// TwinCAT 3 PLC project PRG_B_IO
// Title: B_IO
// Company: RafalOS
// Author: Rafał Osajda
// ProjectVersion: 0.0.0.5
// ProgramVersion: 3.1.4024.0
// libraries:
//   B_Base, * (RafalOS)
//   Tc2_Standard, * (Beckhoff Automation GmbH)
//   Tc2_System, * (Beckhoff Automation GmbH)
//   Tc3_Module, * (Beckhoff Automation GmbH)
// project tree:
//   / PlcTask.TcTTO
//   POUs Compilation/ PRG_Compilation.TcPOU
//   POUs/Electrovalve/ E_ElectrovalveAction.TcDUT, E_ElectrovalveType.TcDUT, FB_Electrovalve.TcPOU, FB_Electrovalve_3on2_NC.TcPOU, FB_Electrovalve_3on2_NO.TcPOU, FB_Electrovalve_5on2_1Coil.TcPOU, FB_Electrovalve_5on2_2Coil.TcPOU, FB_Electrovalve_5on3_2Coil_Vented.TcPOU, FB_Electrovalve_5on3_2Coil_Infected.TcPOU, ITF_Electrovalve.TcIO, ITF_Electrovalve_HMI_Init.TcIO, ITF_Electrovalve_HMI_Connector.TcIO
//   POUs/Sensor/ E_SensorType.TcDUT, FB_Sensor.TcPOU, FB_Sensor_NC.TcPOU, FB_Sensor_NO.TcPOU, FB_Sensor_NO_2InRow.TcPOU, ITF_Sensor.TcIO, ITF_Sensor_HMI_Init.TcIO, ITF_Sensor_HMI_Connector.TcIO
//   POUs/LampkaRozszerzona/ FB_LampBlinking.TcPOU, ITF_LampBlinking.TcIO
//   POUs/Lampka/ FB_Lamp.TcPOU, ITF_Lamp.TcIO
//   POUs/Przyciski/ FB_Button.TcPOU, FB_Button_NC.TcPOU, FB_Button_NO.TcPOU, ITF_Button.TcIO
// real-time tasks:
//   TASK PlcTask: cycle T#10ms, priority 20, ADS port 350

CONFIGURATION PRG_B_IO
    RESOURCE PLC ON TwinCAT3
        TASK PlcTask(INTERVAL := T#10ms, PRIORITY := 20);
        PROGRAM PRG_Compilation WITH PlcTask : PRG_Compilation;
    END_RESOURCE
END_CONFIGURATION

// ---- POUs/Electrovalve/E_ElectrovalveAction.TcDUT
{attribute 'qualified_only'}
{attribute 'strict'}
TYPE E_ElectrovalveAction :
(
	e_EV_Out4_Deactive 	:= 1,
	e_EV_OUT4_Active	:= 2,
	e_EV_Out2_Deactive 	:= 3,
	e_EV_Out2_Active	:= 4,
	e_EV_ToStart		:= 5,
	e_EV_ToEnd			:= 6,
	e_EV_Stop			:= 7,
	e_EV_Reset			:= 8,
	e_EV_Active			:= 9,
	e_EV_Deactive		:= 10
);
END_TYPE

// ---- POUs/Electrovalve/E_ElectrovalveType.TcDUT
{attribute 'qualified_only'}
{attribute 'strict'}
TYPE E_ElectrovalveType :
(
	NC_3na2 	:= 0,
	NO_3na2		:= 1,
	C1_5na2		:= 2,
	C2_5na2		:= 3,
	C2_5na3O	:= 4,	//odpowietrzony
	C2_5na3Z	:= 5	//Zapowietrzony
);
END_TYPE

// ---- POUs/Sensor/E_SensorType.TcDUT
{attribute 'qualified_only'}
{attribute 'strict'}
TYPE E_SensorType :
(
	NO 		:= 0,
	NC		:= 1,
	NOx2	:= 2
);
END_TYPE

// ---- POUs/Sensor/ITF_Sensor.TcIO
(*			
	EVERDE sp. z o.o.
	Rafał Osajda		22.01.2025		TC 4026.13		wer. 0.0.0.1
	B_Baza dla czujników binarnych 	
*)
INTERFACE ITF_Sensor EXTENDS ITF_BaseComponent

(*			
	EVERDE sp. z o.o.
	Rafał Osajda		05.02.2025		TC 4026.13		wer. 0.0.0.1
	Zwraca aktualny stan czujnika
*)
METHOD IsActive : BOOL
END_METHOD

END_INTERFACE

// ---- POUs/Sensor/ITF_Sensor_HMI_Init.TcIO
(*			
	EVERDE sp. z o.o.
	Rafał Osajda		21.08.2025		TC 4024.66
	Interfejs łaczący na potrzeby przekazania do elementu
*)
INTERFACE ITF_Sensor_HMI_Init EXTENDS ITF_BaseComponent, ITF_Sensor_HMI_Connector

END_INTERFACE

// ---- POUs/Sensor/ITF_Sensor_HMI_Connector.TcIO
INTERFACE ITF_Sensor_HMI_Connector EXTENDS ITF_BaseComponent_HMI_Connector

METHOD PUBLIC GetSensorType : E_SensorType
VAR_INPUT
END_VAR
END_METHOD

METHOD PUBLIC GetSensorTypeToString : STRING
END_METHOD

(*			
	EVERDE sp. z o.o.
	Rafał Osajda		05.02.2025		TC 4026.13		wer. 0.0.0.1
	Zwraca aktualny stan czujnika
*)
METHOD IsActive : BOOL
END_METHOD

END_INTERFACE

// ---- POUs/Electrovalve/ITF_Electrovalve.TcIO
(*
	RJM Maszyny sp. z o.o.
	autor 	: Rafał Osajda
	data	: 21.02.2024
	TC		: 3.1 4024.54
	wersja	: 0.0.1.0	: pełna obsługa

	Obsługa elektrozaworu do sterowania siłownikiem pneumatycznym
*)
INTERFACE ITF_Electrovalve EXTENDS ITF_BaseComponent

(*
	RJM Maszyny sp. z o.o.
	autor 	: Rafał Osajda
	data	: 21.02.2024
	TC		: 3.1 4024.54
	wersja	: 0.0.1.0	: pełna obsługa

	Ustawienie odpowiednich wyjść
*)
METHOD Contol : BOOL
VAR_INPUT
	eAction									: E_ElectrovalveAction;
END_VAR
END_METHOD

END_INTERFACE

// ---- POUs/Electrovalve/ITF_Electrovalve_HMI_Init.TcIO
(*			
	EVERDE sp. z o.o.
	Rafał Osajda		21.08.2025		TC 4024.66
	Interfejs łaczący na potrzeby przekazania do elementu
*)
INTERFACE ITF_Electrovalve_HMI_Init EXTENDS ITF_BaseComponent, ITF_Electrovalve_HMI_Connector

END_INTERFACE

// ---- POUs/Electrovalve/ITF_Electrovalve_HMI_Connector.TcIO
INTERFACE ITF_Electrovalve_HMI_Connector EXTENDS ITF_BaseComponent_HMI_Connector

METHOD PUBLIC GetElectrovalveType : E_ElectrovalveType
VAR_INPUT
END_VAR
END_METHOD

METHOD PUBLIC GetElectrovalveTypeToString : STRING
END_METHOD

METHOD IsActiveCoilA : BOOL
VAR_INPUT
END_VAR
END_METHOD

METHOD IsActiveCoilB : BOOL
VAR_INPUT
END_VAR
END_METHOD

END_INTERFACE

// ---- POUs/LampkaRozszerzona/ITF_LampBlinking.TcIO
INTERFACE ITF_LampBlinking EXTENDS ITF_Lamp

(*			
	EVERDE sp. z o.o.
	Rafał Osajda		31.01.2025		TC 4026.13		wer. 0.0.0.1
	Sterowanie działem ipulsatora 
*)
METHOD PUBLIC SetBlink
VAR_INPUT
	bIN				: bool;
END_VAR
END_METHOD

(*			
	EVERDE sp. z o.o.
	Rafał Osajda		31.01.2025		TC 4026.13		wer. 0.0.0.1
	Ustawia czas zgaszonej lampki
*)
METHOD PUBLIC SetTimeOff
VAR_INPUT
	rIN					: REAL;
END_VAR
END_METHOD

(*			
	EVERDE sp. z o.o.
	Rafał Osajda		31.01.2025		TC 4026.13		wer. 0.0.0.1
	
*)
METHOD PUBLIC SetTimeOn
VAR_INPUT
	rIN						: REAL;
END_VAR
END_METHOD

METHOD PUBLIC SetWork
VAR_INPUT
	bShine		: BOOL;
	bBlink		: BOOL;
	rTimeOn		: REAL;
	rTimeOff	: REAL;
END_VAR
END_METHOD

END_INTERFACE

// ---- POUs/Lampka/ITF_Lamp.TcIO
INTERFACE ITF_Lamp EXTENDS ITF_BaseComponent

(*			
	EVERDE sp. z o.o.
	Rafał Osajda		05.02.2025		TC 4026.13		wer. 0.0.0.1
	Sterowanie swieceniem lampki - włącz/wyłącz
*)
METHOD Control
VAR_INPUT
	bIN						: BOOL;
END_VAR
END_METHOD

(*			
	EVERDE sp. z o.o.
	Rafał Osajda		05.02.2025		TC 4026.13		wer. 0.0.0.1
	Zwraca czy lampka wlaczona
*)
METHOD IsActive : BOOL
END_METHOD

(*			
	EVERDE sp. z o.o.
	Rafał Osajda		05.02.2025		TC 4026.13		wer. 0.0.0.1
	Wylacza lampke
*)
METHOD SetOff
END_METHOD

(*			
	EVERDE sp. z o.o.
	Rafał Osajda		05.02.2025		TC 4026.13		wer. 0.0.0.1
	Wlacza lampke
*)
METHOD SetOn
END_METHOD

END_INTERFACE

// ---- POUs/Przyciski/ITF_Button.TcIO
INTERFACE ITF_Button EXTENDS ITF_BaseComponent

METHOD PUBLIC GetRisingEdgePressed : BOOL
VAR_INPUT
END_VAR
END_METHOD

(*			
	EVERDE sp. z o.o.
	Rafał Osajda		31.01.2025		TC 4026.13		wer. 0.0.0.1
	Zwraca stan przycisku
*)
METHOD IsPressed : BOOL
END_METHOD

END_INTERFACE

// ---- POUs Compilation/PRG_Compilation.TcPOU
PROGRAM PRG_Compilation
VAR
	fbCzujnikNC					: FB_Sensor_NC;
	fbCzujnikNO					: FB_Sensor_NO;
	fbCzujnik2xNO				: FB_Sensor_NO_2InRow;
	fbELekrozawor3na2_NC		: FB_Electrovalve_3on2_NC;
	fbELekrozawor3na2_NO		: FB_Electrovalve_3on2_NO;
	fbELekrozawor5na2_1C		: FB_Electrovalve_5on2_1Coil;
	fbELekrozawor5na2_2C		: FB_Electrovalve_5on2_2Coil;
	fbELekrozawor5na2_2C_Odp	: FB_Electrovalve_5on3_2Coil_Vented;
	fbELekrozawor5na2_2C_Zap	: FB_Electrovalve_5on3_2Coil_Infected;
	fbLampka					: FB_Lamp;
	fbLampkaRozszerzona			: FB_LampBlinking;
	fbPrzyciskNC				: FB_Button_NC;
	fbPrzyciskNO				: FB_Button_NO;
END_VAR

END_PROGRAM

// ---- POUs/Sensor/FB_Sensor_NC.TcPOU
(*			
	EVERDE sp. z o.o.
	Rafał Osajda		22.01.2025		TC 4026.13		wer. 0.0.0.1
	B_Baza dla czujników binarnych styk normalnie zamkniety 	
*)
FUNCTION_BLOCK FB_Sensor_NC EXTENDS FB_Sensor
VAR
END_VAR

METHOD FB_init : BOOL
VAR_INPUT
	bInitRetains : BOOL; // if TRUE, the retain variables are initialized (warm start / cold start)
	bInCopyCode : BOOL;  // if TRUE, the instance afterwards gets moved into the copy code (online change)
END_VAR
THIS^.eType		:= E_SensorType.NC;
END_METHOD

(*			
	EVERDE sp. z o.o.
	Rafał Osajda		05.02.2025		TC 4026.13		wer. 0.0.0.1
	Zwraca aktualny stan czujnika
*)
METHOD IsActive : BOOL
IsActive				:= NOT THIS^.bContact;
END_METHOD

END_FUNCTION_BLOCK

// ---- POUs/Sensor/FB_Sensor.TcPOU
(*			
	EVERDE sp. z o.o.
	Rafał Osajda		22.01.2025		TC 4026.13		wer. 0.0.0.1
	B_Baza dla czujników binarnych 	
*)
FUNCTION_BLOCK INTERNAL ABSTRACT FB_Sensor EXTENDS FB_BaseComponent IMPLEMENTS ITF_Sensor, ITF_Sensor_HMI_Init
VAR
	bContact				AT %I*	: BOOL;		// Styk czujnika
	eType							: E_SensorType;
END_VAR

METHOD PUBLIC GetSensorType : E_SensorType
VAR_INPUT
END_VAR
GetSensorType			:= THIS^.eType;
END_METHOD

METHOD PUBLIC GetSensorTypeToString : STRING
VAR CONSTANT
	arrType		: ARRAY [0..2] OF STRING := ['NO', 'NC', 'NOx2'];
END_VAR
GetSensorTypeToString			:= arrType [TO_INT (THIS^.eType)];
END_METHOD

(*			
	EVERDE sp. z o.o.
	Rafał Osajda		05.02.2025		TC 4026.13		wer. 0.0.0.1
	Zwraca aktualny stan czujnika
*)
METHOD IsActive : BOOL
END_METHOD

END_FUNCTION_BLOCK

// ---- POUs/Sensor/FB_Sensor_NO.TcPOU
(*			
	EVERDE sp. z o.o.
	Rafał Osajda		22.01.2025		TC 4026.13		wer. 0.0.0.1
	B_Baza dla czujników binarnych styk normalnie otwarty 	
*)
FUNCTION_BLOCK FB_Sensor_NO EXTENDS FB_Sensor
VAR
END_VAR

METHOD FB_init : BOOL
VAR_INPUT
	bInitRetains : BOOL; // if TRUE, the retain variables are initialized (warm start / cold start)
	bInCopyCode : BOOL;  // if TRUE, the instance afterwards gets moved into the copy code (online change)
END_VAR
THIS^.eType		:= E_SensorType.NO;
END_METHOD

(*			
	EVERDE sp. z o.o.
	Rafał Osajda		05.02.2025		TC 4026.13		wer. 0.0.0.1
	Zwraca aktualny stan czujnika
*)
METHOD IsActive : BOOL
IsActive			:= THIS^.bContact;
END_METHOD

END_FUNCTION_BLOCK

// ---- POUs/Sensor/FB_Sensor_NO_2InRow.TcPOU
(*
	EVERDE sp. z o.o.
	Rafał Osajda
	18.09.2024
	TC3 4026.10
	Obsługa czujników cyforwych NO połączonych szerogowo
*)
FUNCTION_BLOCK FB_Sensor_NO_2InRow EXTENDS FB_Sensor_NO
VAR
	bContact2							AT %I*	: BOOL;		//fizyczne wejście z czujnika
END_VAR

METHOD FB_init : BOOL
VAR_INPUT
	bInitRetains : BOOL; // if TRUE, the retain variables are initialized (warm start / cold start)
	bInCopyCode : BOOL;  // if TRUE, the instance afterwards gets moved into the copy code (online change)
END_VAR
THIS^.eType		:= E_SensorType.NOx2;
END_METHOD

(*			
	EVERDE sp. z o.o.
	Rafał Osajda		05.02.2025		TC 4026.13		wer. 0.0.0.1
	Zwraca aktualny stan czujnika
*)
METHOD IsActive : BOOL
IsActive				:=  THIS^.bContact AND THIS^.bContact2;
END_METHOD

END_FUNCTION_BLOCK

// ---- POUs/Electrovalve/FB_Electrovalve_3on2_NC.TcPOU
(*
	RJM Maszyny sp. z o.o.
	autor 	: Rafał Osajda
	data	: 02.02.2024
	TC		: 3.1 4024.54
	wersja	: 0.0.1.0	: pełna obsługa

	Obsługa elektrozaworu NC
*)
FUNCTION_BLOCK FB_Electrovalve_3on2_NC EXTENDS FB_Electrovalve
VAR
END_VAR

(*
	RJM Maszyny sp. z o.o.
	autor 	: Rafał Osajda
	data	: 21.02.2024
	TC		: 3.1 4024.54
	wersja	: 0.0.1.0	: pełna obsługa

	Ustawienie odpowiednich wyjść
*)METHOD Contol : BOOL
VAR_INPUT
	eAction	: E_ElectrovalveAction;
END_VAR
CASE eAction OF
	E_ElectrovalveAction.e_EV_Out4_Deactive	:
		bCoilA								:= FALSE;
	E_ElectrovalveAction.e_EV_OUT4_Active	:
		bCoilA								:= TRUE;
	E_ElectrovalveAction.e_EV_Reset			:
		bCoilA								:= FALSE;

END_CASE
bCoilB										:= FALSE;
END_METHOD

METHOD FB_init : BOOL
VAR_INPUT
	bInitRetains : BOOL; // if TRUE, the retain variables are initialized (warm start / cold start)
	bInCopyCode : BOOL;  // if TRUE, the instance afterwards gets moved into the copy code (online change)
END_VAR
THIS^.eType			:= E_ElectrovalveType.NC_3na2;
END_METHOD

END_FUNCTION_BLOCK

// ---- POUs/Electrovalve/FB_Electrovalve.TcPOU
(*
	RJM Maszyny sp. z o.o.
	autor 	: Rafał Osajda
	data	: 02.02.2024
	TC		: 3.1 4024.54
	wersja	: 0.0.1.0	: pełna obsługa

	Obsługa elektrozaworu do sterowania siłownikiem pneumatycznym. FB bazowy dla pozostałych rodzajów elektrozaworów
*)
FUNCTION_BLOCK ABSTRACT FB_Electrovalve EXTENDS FB_BaseComponent IMPLEMENTS  ITF_Electrovalve, ITF_Electrovalve_HMI_Init
VAR
	bCoilA							AT %Q*	: BOOL;
	bCoilB							AT %Q*	: BOOL;
	eType									: E_ElectrovalveType;
END_VAR

(*
	RJM Maszyny sp. z o.o.
	autor 	: Rafał Osajda
	data	: 21.02.2024
	TC		: 3.1 4024.54
	wersja	: 0.0.1.0	: pełna obsługa

	Ustawienie odpowiednich wyjść
*)
METHOD Contol : BOOL
VAR_INPUT
	eAction	: E_ElectrovalveAction;
END_VAR
END_METHOD

METHOD PUBLIC GetElectrovalveType : E_ElectrovalveType
VAR_INPUT
END_VAR
GetElectrovalveType			:= THIS^.eType;
END_METHOD

METHOD PUBLIC GetElectrovalveTypeToString : STRING
VAR CONSTANT
	arrType		: ARRAY [0..5] OF STRING := ['NC_3na2', 'NO_3na2', 'C1_5na2', 'C2_5na2', 'C2_5na3O', 'C2_5na3Z'];
END_VAR
GetElectrovalveTypeToString			:= arrType [TO_INT (THIS^.eType)];
END_METHOD

METHOD IsActiveCoilA : BOOL
VAR_INPUT
END_VAR
IsActiveCoilA			:= THIS^.bCoilA;
END_METHOD

METHOD IsActiveCoilB : BOOL
VAR_INPUT
END_VAR
IsActiveCoilB			:= THIS^.bCoilB;
END_METHOD

END_FUNCTION_BLOCK

// ---- POUs/Electrovalve/FB_Electrovalve_3on2_NO.TcPOU
(*
	RJM Maszyny sp. z o.o.
	autor 	: Rafał Osajda
	data	: 02.02.2024
	TC		: 3.1 4024.54
	wersja	: 0.0.1.0	: pełna obsługa

	Obsługa elektrozaworu NO
*)
FUNCTION_BLOCK FB_Electrovalve_3on2_NO EXTENDS FB_Electrovalve
VAR
END_VAR

(*
	RJM Maszyny sp. z o.o.
	autor 	: Rafał Osajda
	data	: 21.02.2024
	TC		: 3.1 4024.54
	wersja	: 0.0.1.0	: pełna obsługa

	Ustawienie odpowiednich wyjść
*)
METHOD Contol : BOOL
VAR_INPUT
	eAction	: E_ElectrovalveAction;
END_VAR
CASE eAction OF
	E_ElectrovalveAction.e_EV_Out4_Deactive	:
		bCoilA								:= TRUE;
	E_ElectrovalveAction.e_EV_OUT4_Active	:
		bCoilA								:= FALSE;
	E_ElectrovalveAction.e_EV_Reset			:
		bCoilA								:= FALSE;

END_CASE
bCoilB										:= FALSE;
END_METHOD

METHOD FB_init : BOOL
VAR_INPUT
	bInitRetains : BOOL; // if TRUE, the retain variables are initialized (warm start / cold start)
	bInCopyCode : BOOL;  // if TRUE, the instance afterwards gets moved into the copy code (online change)
END_VAR
THIS^.eType			:= E_ElectrovalveType.NO_3na2;
END_METHOD

END_FUNCTION_BLOCK

// ---- POUs/Electrovalve/FB_Electrovalve_5on2_1Coil.TcPOU
(*
	RJM Maszyny sp. z o.o.
	autor 	: Rafał Osajda
	data	: 02.02.2024
	TC		: 3.1 4024.54
	wersja	: 0.0.1.0	: pełna obsługa

	Obsługa elektrozaworu do sterowania siłownikiem pneumatycznym.sterowanie 5 na 2 1 cewka
*)
FUNCTION_BLOCK FB_Electrovalve_5on2_1Coil EXTENDS FB_Electrovalve

(*
	RJM Maszyny sp. z o.o.
	autor 	: Rafał Osajda
	data	: 21.02.2024
	TC		: 3.1 4024.54
	wersja	: 0.0.1.0	: pełna obsługa

	Ustawienie odpowiednich wyjść
*)
METHOD Contol : BOOL
VAR_INPUT
	eAction	: E_ElectrovalveAction;
END_VAR
CASE eAction OF
	E_ElectrovalveAction.e_EV_Out4_Deactive	:
		bCoilA								:= FALSE;
	E_ElectrovalveAction.e_EV_OUT4_Active	:
		bCoilA								:= TRUE;
	E_ElectrovalveAction.e_EV_ToStart	:
		bCoilA								:= FALSE;
	E_ElectrovalveAction.e_EV_ToEnd		:
		bCoilA								:= TRUE;
	E_ElectrovalveAction.e_EV_Reset			:
		bCoilA								:= FALSE;
END_CASE
THIS^.bCoilB								:= FALSE;
END_METHOD

METHOD FB_init : BOOL
VAR_INPUT
	bInitRetains : BOOL; // if TRUE, the retain variables are initialized (warm start / cold start)
	bInCopyCode : BOOL;  // if TRUE, the instance afterwards gets moved into the copy code (online change)
END_VAR
THIS^.eType			:= E_ElectrovalveType.C1_5na2;
END_METHOD

END_FUNCTION_BLOCK

// ---- POUs/Electrovalve/FB_Electrovalve_5on2_2Coil.TcPOU
(*
	RJM Maszyny sp. z o.o.
	autor 	: Rafał Osajda
	data	: 02.02.2024
	TC		: 3.1 4024.54
	wersja	: 0.0.1.0	: pełna obsługa

	Obsługa elektrozaworu do sterowania siłownikiem pneumatycznym.sterowanie 5 na 2 2 cewki
*)
FUNCTION_BLOCK FB_Electrovalve_5on2_2Coil EXTENDS FB_Electrovalve

(*
	RJM Maszyny sp. z o.o.
	autor 	: Rafał Osajda
	data	: 21.02.2024
	TC		: 3.1 4024.54
	wersja	: 0.0.1.0	: pełna obsługa

	Ustawienie odpowiednich wyjść
*)
METHOD Contol : BOOL
VAR_INPUT
	eAction									: E_ElectrovalveAction;
END_VAR
CASE eAction OF
	E_ElectrovalveAction.e_EV_Out4_Deactive	:
		bCoilA								:= FALSE;
	E_ElectrovalveAction.e_EV_OUT4_Active	:
		bCoilA								:= TRUE;
		bCoilB								:= FALSE;
	E_ElectrovalveAction.e_EV_Out2_Deactive	:
		bCoilB								:= FALSE;
	E_ElectrovalveAction.e_EV_Out2_Active	:
		bCoilB								:= TRUE;
		bCoilA								:= FALSE;
	E_ElectrovalveAction.e_EV_ToStart	:
		bCoilA								:= FALSE;
		bCoilB								:= TRUE;
	E_ElectrovalveAction.e_EV_ToEnd		:
		bCoilA								:= TRUE;
		bCoilB								:= FALSE;
	E_ElectrovalveAction.e_EV_Reset			:
		bCoilA								:= FALSE;
		bCoilB								:= FALSE;
	E_ElectrovalveAction.e_EV_Active			:
		bCoilA								:= TRUE;
		bCoilB								:= TRUE;
	E_ElectrovalveAction.e_EV_Deactive		:
		bCoilA								:= FALSE;
		bCoilB								:= FALSE;	
END_CASE
END_METHOD

METHOD FB_init : BOOL
VAR_INPUT
	bInitRetains : BOOL; // if TRUE, the retain variables are initialized (warm start / cold start)
	bInCopyCode : BOOL;  // if TRUE, the instance afterwards gets moved into the copy code (online change)
END_VAR
THIS^.eType			:= E_ElectrovalveType.C2_5na2;
END_METHOD

END_FUNCTION_BLOCK

// ---- POUs/Electrovalve/FB_Electrovalve_5on3_2Coil_Vented.TcPOU
(*
	RJM Maszyny sp. z o.o.
	autor 	: Rafał Osajda
	data	: 02.02.2024
	TC		: 3.1 4024.54
	wersja	: 0.0.1.0	: pełna obsługa

	Obsługa elektrozaworu do sterowania siłownikiem pneumatycznym.sterowanie 5 na 3 2 cewki odpowietrzone
*)
FUNCTION_BLOCK FB_Electrovalve_5on3_2Coil_Vented EXTENDS FB_Electrovalve

(*
	RJM Maszyny sp. z o.o.
	autor 	: Rafał Osajda
	data	: 21.02.2024
	TC		: 3.1 4024.54
	wersja	: 0.0.1.0	: pełna obsługa

	Ustawienie odpowiednich wyjść
*)
METHOD Contol : BOOL
VAR_INPUT
	eAction									: E_ElectrovalveAction;
END_VAR
CASE eAction OF
	E_ElectrovalveAction.e_EV_Out4_Deactive	:
		bCoilA								:= FALSE;
	E_ElectrovalveAction.e_EV_OUT4_Active	:
		bCoilA								:= TRUE;
	E_ElectrovalveAction.e_EV_Out2_Deactive	:
		bCoilB								:= FALSE;
	E_ElectrovalveAction.e_EV_Out2_Active	:
		bCoilB								:= TRUE;
	E_ElectrovalveAction.e_EV_ToStart	:
		bCoilA								:= FALSE;
		bCoilB								:= TRUE;
	E_ElectrovalveAction.e_EV_ToEnd		:
		bCoilA								:= TRUE;
		bCoilB								:= FALSE;
	E_ElectrovalveAction.e_EV_Stop		:
		bCoilA								:= TRUE;
		bCoilB								:= TRUE;
	E_ElectrovalveAction.e_EV_Reset			:
		bCoilA								:= FALSE;
		bCoilB								:= FALSE;
	E_ElectrovalveAction.e_EV_Active			:
		bCoilA								:= TRUE;
		bCoilB								:= TRUE;
	E_ElectrovalveAction.e_EV_Deactive		:
		bCoilA								:= FALSE;
		bCoilB								:= FALSE;		
END_CASE
END_METHOD

METHOD FB_init : BOOL
VAR_INPUT
	bInitRetains : BOOL; // if TRUE, the retain variables are initialized (warm start / cold start)
	bInCopyCode : BOOL;  // if TRUE, the instance afterwards gets moved into the copy code (online change)
END_VAR
THIS^.eType			:= E_ElectrovalveType.C2_5na3O;
END_METHOD

END_FUNCTION_BLOCK

// ---- POUs/Electrovalve/FB_Electrovalve_5on3_2Coil_Infected.TcPOU
(*
	RJM Maszyny sp. z o.o.
	autor 	: Rafał Osajda
	data	: 02.02.2024
	TC		: 3.1 4024.54
	wersja	: 0.0.1.0	: pełna obsługa

	Obsługa elektrozaworu do sterowania siłownikiem pneumatycznym.sterowanie 5 na 3 2 cewki zapowietrzone
*)
FUNCTION_BLOCK FB_Electrovalve_5on3_2Coil_Infected EXTENDS FB_Electrovalve

(*
	RJM Maszyny sp. z o.o.
	autor 	: Rafał Osajda
	data	: 21.02.2024
	TC		: 3.1 4024.54
	wersja	: 0.0.1.0	: pełna obsługa

	Ustawienie odpowiednich wyjść
*)
METHOD Contol : BOOL
VAR_INPUT
	eAction									: E_ElectrovalveAction;
END_VAR
CASE eAction OF
	E_ElectrovalveAction.e_EV_Out4_Deactive	:
		bCoilA								:= TRUE;
	E_ElectrovalveAction.e_EV_OUT4_Active	:
		bCoilA								:= FALSE;
	E_ElectrovalveAction.e_EV_Out2_Deactive	:
		bCoilB								:= TRUE;
	E_ElectrovalveAction.e_EV_Out2_Active	:
		bCoilB								:= FALSE;
	E_ElectrovalveAction.e_EV_ToStart	:
		bCoilA								:= TRUE;
		bCoilB								:= FALSE;
	E_ElectrovalveAction.e_EV_ToEnd		:
		bCoilA								:= FALSE;
		bCoilB								:= TRUE;
	E_ElectrovalveAction.e_EV_Stop		:
		bCoilA								:= FALSE;
		bCoilB								:= FALSE;
	E_ElectrovalveAction.e_EV_Reset			:
		bCoilA								:= FALSE;
		bCoilB								:= FALSE;
	E_ElectrovalveAction.e_EV_Active			:
		bCoilA								:= FALSE;
		bCoilB								:= FALSE;
	E_ElectrovalveAction.e_EV_Deactive		:
		bCoilA								:= FALSE;
		bCoilB								:= FALSE;	
END_CASE
END_METHOD

METHOD FB_init : BOOL
VAR_INPUT
	bInitRetains : BOOL; // if TRUE, the retain variables are initialized (warm start / cold start)
	bInCopyCode : BOOL;  // if TRUE, the instance afterwards gets moved into the copy code (online change)
END_VAR
THIS^.eType			:= E_ElectrovalveType.C2_5na3Z;
END_METHOD

END_FUNCTION_BLOCK

// ---- POUs/Lampka/FB_Lamp.TcPOU
(*			
	EVERDE sp. z o.o.
	Rafał Osajda		22.01.2025		TC 4026.13		wer. 0.0.0.1
	Sterowanie lampką
*)
FUNCTION_BLOCK FB_Lamp EXTENDS FB_BaseComponent IMPLEMENTS ITF_Lamp
VAR
	bOut							AT %Q*	: BOOL;		// Lampka
END_VAR

(*			
	EVERDE sp. z o.o.
	Rafał Osajda		05.02.2025		TC 4026.13		wer. 0.0.0.1
	Sterowanie swieceniem lampki - włącz/wyłącz
*)
METHOD Control
VAR_INPUT
	bIN	: BOOL;
END_VAR
IF (bIN) THEN
	THIS^.SetOn ();
ELSE
	THIS^.SetOff ();
END_IF
END_METHOD

(*			
	EVERDE sp. z o.o.
	Rafał Osajda		05.02.2025		TC 4026.13		wer. 0.0.0.1
	Zwraca czy lampka wlaczona
*)
METHOD IsActive : BOOL
IsActive					:= THIS^.bOut;
END_METHOD

(*			
	EVERDE sp. z o.o.
	Rafał Osajda		05.02.2025		TC 4026.13		wer. 0.0.0.1
	Wylacza lampke
*)
METHOD SetOff
THIS^.bOut				:= FALSE;
END_METHOD

(*			
	EVERDE sp. z o.o.
	Rafał Osajda		05.02.2025		TC 4026.13		wer. 0.0.0.1
	Wlacza lampke
*)
METHOD SetOn
THIS^.bOut				:= TRUE;
END_METHOD

END_FUNCTION_BLOCK

// ---- POUs/LampkaRozszerzona/FB_LampBlinking.TcPOU
(*			
	EVERDE sp. z o.o.
	Rafał Osajda		16.07.2025		TC 4024.66
	Lampka rozszerzona o moduł FB_Impuls co integruje w niej możlwiość mgania lub świecenie ciągłego
*)
FUNCTION_BLOCK FB_LampBlinking EXTENDS FB_Lamp IMPLEMENTS ITF_LampBlinking
VAR
	fbImpulse				: FB_BaseImpulse;
END_VAR

(*			
	EVERDE sp. z o.o.
	Rafał Osajda		05.02.2025		TC 4026.13		wer. 0.0.0.1
	Sterowanie swieceniem lampki - włącz/wyłącz
*)
METHOD Control
VAR_INPUT
	bIN	: BOOL;
END_VAR
IF (bIN) THEN
	THIS^.fbImpulse.SetExecuteOn ();
ELSE
	THIS^.fbImpulse.SetExecuteOff ();
END_IF
END_METHOD

(*			
	EVERDE sp. z o.o.
	Rafał Osajda		27.03.2025		TC 4024.66
	Wywolanie co cykl operacji 
*)
METHOD PUBLIC ExecuteEveryCycle_Operation
VAR_INPUT
END_VAR
SUPER^.ExecuteEveryCycle_Operation ();

THIS^.fbImpulse ();
END_METHOD

(*			
	EVERDE sp. z o.o.
	Rafał Osajda		27.03.2025		TC 4024.66
	Aktualizacja flag 
*)
METHOD PUBLIC ExecuteEveryCycle_Status
VAR_INST
END_VAR
SUPER^.ExecuteEveryCycle_Status ();

THIS^.bOut		:= THIS^.fbImpulse.GetExit ();
END_METHOD

(*			
	EVERDE sp. z o.o.
	Rafał Osajda		31.01.2025		TC 4026.13		wer. 0.0.0.1
	Sterowanie działem ipulsatora 
*)
METHOD PUBLIC SetBlink
VAR_INPUT
	bIN				: bool;
END_VAR
THIS^.fbImpulse.SetFlashing (bIN	:= bIN);
END_METHOD

(*			
	EVERDE sp. z o.o.
	Rafał Osajda		05.02.2025		TC 4026.13		wer. 0.0.0.1
	Wylacza lampke
*)
METHOD SetOff
THIS^.fbImpulse.SetExecuteOff ();
END_METHOD

(*			
	EVERDE sp. z o.o.
	Rafał Osajda		05.02.2025		TC 4026.13		wer. 0.0.0.1
	Wlacza lampke - praca ciągła
*)
METHOD SetOn
THIS^.fbImpulse.SetExecuteOn ();
END_METHOD

METHOD PUBLIC SetShine
VAR_INPUT
	bIN				: BOOL;
END_VAR
IF (bIN) THEN
	THIS^.fbImpulse.SetExecuteOn ();
ELSE
	THIS^.fbImpulse.SetExecuteOff ();
END_IF
END_METHOD

(*			
	EVERDE sp. z o.o.
	Rafał Osajda		31.01.2025		TC 4026.13		wer. 0.0.0.1
	Ustawia czas zgaszonej lampki
*)
METHOD PUBLIC SetTimeOff
VAR_INPUT
	rIN					: REAL;
END_VAR
THIS^.fbImpulse.SetTimeOff (rIN	:= rIN);
END_METHOD

(*			
	EVERDE sp. z o.o.
	Rafał Osajda		31.01.2025		TC 4026.13		wer. 0.0.0.1
	
*)
METHOD PUBLIC SetTimeOn
VAR_INPUT
	rIN						: REAL;
END_VAR
THIS^.fbImpulse.SetTimeOn (rIN	:= rIN);
END_METHOD

METHOD PUBLIC SetWork
VAR_INPUT
	bShine		: BOOL;
	bBlink		: BOOL;
	rTimeOn		: REAL;
	rTimeOff	: REAL;
END_VAR
THIS^.fbImpulse.SetTimeOn (rIN := rTimeOn);
THIS^.fbImpulse.SetTimeOff (rIN := rTimeOff);
THIS^.SetShine (bIN	:= bShine);
THIS^.SetBlink (bIN := bBlink);
END_METHOD

END_FUNCTION_BLOCK

// ---- POUs/Przyciski/FB_Button_NC.TcPOU
(*			
	EVERDE sp. z o.o.
	Rafał Osajda		31.01.2025		TC 4026.13		wer. 0.0.0.1
	Obsługa przycisku ze stykiem NC
*)
FUNCTION_BLOCK FB_Button_NC EXTENDS FB_Button
VAR
END_VAR

METHOD PUBLIC GetRisingEdgePressed : BOOL
VAR_INPUT
END_VAR
IF (THIS^.bContactPrev AND NOT THIS^.bContact) THEN
	THIS^.bContactPrev		:= FALSE;
	GetRisingEdgePressed	:= TRUE;
ELSIF (NOT THIS^.bContactPrev AND THIS^.bContact) THEN
	THIS^.bContactPrev		:= TRUE;
END_IF
END_METHOD

(*			
	EVERDE sp. z o.o.
	Rafał Osajda		31.01.2025		TC 4026.13		wer. 0.0.0.1
	Zwraca stan przycisku
*)
METHOD IsPressed : BOOL
IsPressed			:= NOT THIS^.bContact;
END_METHOD

END_FUNCTION_BLOCK

// ---- POUs/Przyciski/FB_Button.TcPOU
(*			
	EVERDE sp. z o.o.
	Rafał Osajda		31.01.2025		TC 4026.13		wer. 0.0.0.1
	Obsługa przycisków 
*)
FUNCTION_BLOCK ABSTRACT FB_Button EXTENDS FB_BaseComponent IMPLEMENTS ITF_Button
VAR
	bContact							AT %I*	: BOOL;		// Styk przycisku 
	bContactPrev								: BOOL;
END_VAR

METHOD PUBLIC GetRisingEdgePressed : BOOL
VAR_INPUT
END_VAR
END_METHOD

(*			
	EVERDE sp. z o.o.
	Rafał Osajda		31.01.2025		TC 4026.13		wer. 0.0.0.1
	Zwraca stan przycisku
*)
METHOD IsPressed : BOOL
END_METHOD

END_FUNCTION_BLOCK

// ---- POUs/Przyciski/FB_Button_NO.TcPOU
(*			
	EVERDE sp. z o.o.
	Rafał Osajda		31.01.2025		TC 4026.13		wer. 0.0.0.1
	Obsługa przycisku ze stykiem NO
*)
FUNCTION_BLOCK FB_Button_NO EXTENDS FB_Button
VAR
END_VAR

METHOD PUBLIC GetRisingEdgePressed : BOOL
VAR_INPUT
END_VAR
IF (NOT THIS^.bContactPrev AND THIS^.bContact) THEN
	THIS^.bContactPrev 			:= TRUE;
	GetRisingEdgePressed		:= TRUE;
ELSIF (THIS^.bContactPrev AND NOT THIS^.bContact) THEN
	THIS^.bContactPrev			:= FALSE;
END_IF
END_METHOD

(*			
	EVERDE sp. z o.o.
	Rafał Osajda		31.01.2025		TC 4026.13		wer. 0.0.0.1
	Zwraca stan przycisku
*)
METHOD IsPressed : BOOL
IsPressed			:= THIS^.bContact;
END_METHOD

END_FUNCTION_BLOCK
